ABB RAPID module: 00417E3D

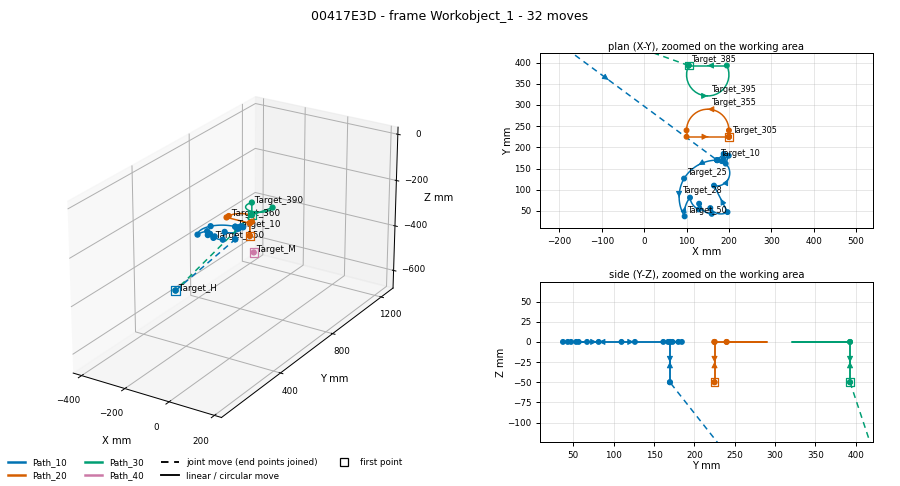
[picture p0: tool path of 00417E3D in frame Workobject_1, 32 of 32 moves have a stored position in this frame; points joined in program order, loops and branches not executed]
MODULE Module1
        CONST robtarget Target_H:=[[-349.999997471,555.651291784,-538.588637673],[0.701057388,-0.092295986,-0.092295969,-0.701057375],[0,0,0,0],[9E+09,9E+09,9E+09,9E+09,9E+09,9E+09]];
    CONST robtarget Target_10:=[[172.145654378,169.721037846,0],[0.015654757,0,0,0.999877457],[1,-2,1,0],[9E+09,9E+09,9E+09,9E+09,9E+09,9E+09]];
    CONST robtarget Target_20:=[[127.176015411,158.806349071,0],[0.015654757,0,0,0.999877457],[1,-2,1,0],[9E+09,9E+09,9E+09,9E+09,9E+09,9E+09]];
    CONST robtarget Target_30:=[[94.179068929,126.362545613,0],[0.015654757,0,0,0.999877457],[1,-2,1,0],[9E+09,9E+09,9E+09,9E+09,9E+09,9E+09]];
    CONST robtarget Target_40:=[[82.505775243,81.583833322,0],[0.015654757,0,0,0.999877457],[1,-2,1,0],[9E+09,9E+09,9E+09,9E+09,9E+09,9E+09]];
    CONST robtarget Target_50:=[[95.464213358,37.159991282,0],[0.015654757,0,0,0.999877457],[1,-2,1,0],[9E+09,9E+09,9E+09,9E+09,9E+09,9E+09]];
    CONST robtarget Target_60:=[[108.140548997,81.368919049,0],[0.015654757,0,0,0.999877457],[1,-2,1,0],[9E+09,9E+09,9E+09,9E+09,9E+09,9E+09]];
    CONST robtarget Target_70:=[[99.986563128,67.9517476,0],[0.015654757,0,0,0.999877457],[1,-2,1,0],[9E+09,9E+09,9E+09,9E+09,9E+09,9E+09]];
    CONST robtarget Target_80:=[[115.844,63.278,0],[0.015654757,0,0,0.999877457],[1,-2,1,0],[9E+09,9E+09,9E+09,9E+09,9E+09,9E+09]];
    CONST robtarget Target_90:=[[110.943419364,69.425655071,0],[0.015654757,0,0,0.999877457],[1,-2,1,0],[9E+09,9E+09,9E+09,9E+09,9E+09,9E+09]];
    CONST robtarget Target_100:=[[118.270530204,59.586392727,0],[0.015654757,0,0,0.999877457],[1,-2,1,0],[9E+09,9E+09,9E+09,9E+09,9E+09,9E+09]];
    CONST robtarget Target_110:=[[128.909818396,53.478759508,0],[0.015654757,0,0,0.999877457],[1,-2,1,0],[9E+09,9E+09,9E+09,9E+09,9E+09,9E+09]];
    CONST robtarget Target_120:=[[129.685602376,67.032677318,0],[0.015654757,0,0,0.999877457],[1,-2,1,0],[9E+09,9E+09,9E+09,9E+09,9E+09,9E+09]];
    CONST robtarget Target_130:=[[135.242270658,54.463630271,0],[0.015654757,0,0,0.999877457],[1,-2,1,0],[9E+09,9E+09,9E+09,9E+09,9E+09,9E+09]];
    CONST robtarget Target_140:=[[145.944316156,45.842509218,0],[0.015654757,0,0,0.999877457],[1,-2,1,0],[9E+09,9E+09,9E+09,9E+09,9E+09,9E+09]];
    CONST robtarget Target_150:=[[159.408253951,43.089350102,0],[0.015654757,0,0,0.999877457],[1,-2,1,0],[9E+09,9E+09,9E+09,9E+09,9E+09,9E+09]];
    CONST robtarget Target_160:=[[156.13873613,56.659281011,0],[0.015654757,0,0,0.999877457],[1,-2,1,0],[9E+09,9E+09,9E+09,9E+09,9E+09,9E+09]];
    CONST robtarget Target_170:=[[167.339659667,46.46756084,0],[0.015654757,0,0,0.999877457],[1,-2,1,0],[9E+09,9E+09,9E+09,9E+09,9E+09,9E+09]];
    CONST robtarget Target_180:=[[156.961,49.601,0],[0.015654757,0,0,0.999877457],[1,-2,1,0],[9E+09,9E+09,9E+09,9E+09,9E+09,9E+09]];
    CONST robtarget Target_190:=[[196.643218036,47.197896671,0],[0.015654757,0,0,0.999877457],[1,-1,1,0],[9E+09,9E+09,9E+09,9E+09,9E+09,9E+09]];
    CONST robtarget Target_200:=[[180.134939682,64.681155269,0],[0.015654757,0,0,0.999877457],[1,-2,1,0],[9E+09,9E+09,9E+09,9E+09,9E+09,9E+09]];
    CONST robtarget Target_210:=[[169.208263421,86.100663464,0],[0.015654757,0,0,0.999877457],[1,-2,1,0],[9E+09,9E+09,9E+09,9E+09,9E+09,9E+09]];
    CONST robtarget Target_220:=[[164.744756678,109.728289095,0],[0.015654757,0,0,0.999877457],[1,-2,1,0],[9E+09,9E+09,9E+09,9E+09,9E+09,9E+09]];
    CONST robtarget Target_230:=[[189.86479429,115.046784411,0],[0.015654757,0,0,0.999877457],[1,-2,1,0],[9E+09,9E+09,9E+09,9E+09,9E+09,9E+09]];
    CONST robtarget Target_240:=[[201.945805105,137.70405388,0],[0.015654757,0,0,0.999877457],[1,-2,1,0],[9E+09,9E+09,9E+09,9E+09,9E+09,9E+09]];
    CONST robtarget Target_250:=[[192.36364797,161.525996428,0],[0.015654757,0,0,0.999877457],[1,-2,1,0],[9E+09,9E+09,9E+09,9E+09,9E+09,9E+09]];
    CONST robtarget Target_260:=[[199.538662434,180.200691671,0],[0.015654757,0,0,0.999877457],[1,-2,1,0],[9E+09,9E+09,9E+09,9E+09,9E+09,9E+09]];
    CONST robtarget Target_270:=[[187.501772235,172.981329375,0],[0.015654757,0,0,0.999877457],[1,-2,1,0],[9E+09,9E+09,9E+09,9E+09,9E+09,9E+09]];
    CONST robtarget Target_280:=[[183.067776679,167.478919652,0],[0.015654757,0,0,0.999877457],[1,-2,1,0],[9E+09,9E+09,9E+09,9E+09,9E+09,9E+09]];
    CONST robtarget Target_290:=[[187.548582623,184.533188144,0],[0.015654757,0,0,0.999877457],[1,-2,1,0],[9E+09,9E+09,9E+09,9E+09,9E+09,9E+09]];
    CONST robtarget Target_300:=[[172.145654378,169.721037846,0],[0.015654757,0,0,0.999877457],[1,-2,1,0],[9E+09,9E+09,9E+09,9E+09,9E+09,9E+09]];
    CONST robtarget Target_305:=[[200,225,-50],[0.015654757,0,0,0.999877457],[1,-2,1,0],[9E+09,9E+09,9E+09,9E+09,9E+09,9E+09]];
    CONST robtarget Target_310:=[[200,225,0],[0.015654757,0,0,0.999877457],[1,-2,1,0],[9E+09,9E+09,9E+09,9E+09,9E+09,9E+09]];
    CONST robtarget Target_320:=[[200,240,0],[0.015654757,0,0,0.999877457],[1,-2,1,0],[9E+09,9E+09,9E+09,9E+09,9E+09,9E+09]];
    CONST robtarget Target_330:=[[185.355339059,275.355339059,0],[0.015654757,0,0,0.999877457],[1,-2,1,0],[9E+09,9E+09,9E+09,9E+09,9E+09,9E+09]];
    CONST robtarget Target_340:=[[150,290,0],[0.015654757,0,0,0.999877457],[1,-2,1,0],[9E+09,9E+09,9E+09,9E+09,9E+09,9E+09]];
    CONST robtarget Target_350:=[[114.644660941,275.355339059,0],[0.015654757,0,0,0.999877457],[1,-2,1,0],[9E+09,9E+09,9E+09,9E+09,9E+09,9E+09]];
    CONST robtarget Target_360:=[[100,240,0],[0.015654757,0,0,0.999877457],[1,-2,1,0],[9E+09,9E+09,9E+09,9E+09,9E+09,9E+09]];
    CONST robtarget Target_370:=[[100,225,0],[0.015654757,0,0,0.999877457],[1,-2,1,0],[9E+09,9E+09,9E+09,9E+09,9E+09,9E+09]];
    CONST robtarget Target_380:=[[200,225,0],[0.015654757,0,0,0.999877457],[1,-2,1,0],[9E+09,9E+09,9E+09,9E+09,9E+09,9E+09]];
    CONST robtarget Target_385:=[[105,392.991805459,-50],[0.015654757,0,0,0.999877457],[1,-2,1,0],[9E+09,9E+09,9E+09,9E+09,9E+09,9E+09]];
    CONST robtarget Target_390:=[[105,392.991805459,0],[0.015654757,0,0,0.999877457],[1,-2,1,0],[9E+09,9E+09,9E+09,9E+09,9E+09,9E+09]];
    CONST robtarget Target_400:=[[103.164813866,353.691159257,0],[0.015654757,0,0,0.999877457],[1,-2,1,0],[9E+09,9E+09,9E+09,9E+09,9E+09,9E+09]];
    CONST robtarget Target_410:=[[130.328264565,325.22968273,0],[0.015654757,0,0,0.999877457],[1,-2,1,0],[9E+09,9E+09,9E+09,9E+09,9E+09,9E+09]];
    CONST robtarget Target_420:=[[169.671735435,325.22968273,0],[0.015654757,0,0,0.999877457],[1,-2,1,0],[9E+09,9E+09,9E+09,9E+09,9E+09,9E+09]];
    CONST robtarget Target_430:=[[196.835186134,353.691159257,0],[0.015654757,0,0,0.999877457],[1,-2,1,0],[9E+09,9E+09,9E+09,9E+09,9E+09,9E+09]];
    CONST robtarget Target_440:=[[195,392.991805459,0],[0.015654757,0,0,0.999877457],[1,-2,1,0],[9E+09,9E+09,9E+09,9E+09,9E+09,9E+09]];
    CONST robtarget Target_M:=[[-410.514648889,1245.713795009,-649.374024814],[0.613768807,0.08026289,-0.406843498,-0.671806585],[0,-1,0,0],[9E+09,9E+09,9E+09,9E+09,9E+09,9E+09]];
    CONST robtarget Target_355:=[[150,290,0],[0.015654757,0,0,0.999877457],[1,-2,1,0],[9E+09,9E+09,9E+09,9E+09,9E+09,9E+09]];
    CONST robtarget Target_15:=[[127.992,158.531,0],[0.015654757,0,0,0.999877457],[1,-2,1,0],[9E+09,9E+09,9E+09,9E+09,9E+09,9E+09]];
    CONST robtarget Target_28:=[[82.508,84.221,0],[0.015654757,0,0,0.999877457],[1,-2,1,0],[9E+09,9E+09,9E+09,9E+09,9E+09,9E+09]];
    CONST robtarget Target_25:=[[94.179,126.363,0],[0.015654757,0,0,0.999877457],[1,-2,1,0],[9E+09,9E+09,9E+09,9E+09,9E+09,9E+09]];
    CONST robtarget Target_395:=[[150,321.197,0],[0.015654757,0,0,0.999877457],[1,-2,1,0],[9E+09,9E+09,9E+09,9E+09,9E+09,9E+09]];
    CONST robtarget Target_55:=[[97.319,60.55,0],[0.015654757,0,0,0.999877457],[1,-2,1,0],[9E+09,9E+09,9E+09,9E+09,9E+09,9E+09]];
    CONST robtarget Target_125:=[[138.21,52.221,0],[0.015654757,0,0,0.999877457],[1,-2,1,0],[9E+09,9E+09,9E+09,9E+09,9E+09,9E+09]];
    CONST robtarget Target_185:=[[167.277,46.352,0],[0.015654757,0,0,0.999877457],[1,-2,1,0],[9E+09,9E+09,9E+09,9E+09,9E+09,9E+09]];
    CONST robtarget Target_115:=[[128.566,60.282,0],[0.015654757,0,0,0.999877457],[0,0,0,0],[9E+09,9E+09,9E+09,9E+09,9E+09,9E+09]];
!***********************************************************
    !
    ! M?dulo:  Module1
    !
    ! Descripción:
    !   <Introduzca la descripción aquí>
    !
    ! Autor: ASUS
    !
    ! Versión: 1.0
    !
    !***********************************************************


    !***********************************************************
    !
    ! Procedimiento Main
    !
    !   Este es el punto de entrada de su programa
    !
    !***********************************************************
    PROC main()
        !Add your code here
        WHILE TRUE DO
            IF DI_01=1 THEN
                set DO_01;
                first;
                Reset DO_01;
            ELSEIF DI_02=1 THEN
                set DO_02;
                Path_40;
                Reset DO_02;
            ENDIF
        ENDWHILE
    ENDPROC
    PROC Path_10()
        MoveJ Target_H,v100,z5,THerramienta\WObj:=Workobject_1;
        MoveJ [[172.145654378,169.721037846,-50],[0.015654757,0,0,0.999877457],[1,-2,1,0],[9E+09,9E+09,9E+09,9E+09,9E+09,9E+09]],v400,z5,THerramienta\WObj:=Workobject_1;
        MoveL Target_10,v200,z0,THerramienta\WObj:=Workobject_1;
        MoveC Target_15,Target_25,v200,z5,THerramienta\WObj:=Workobject_1;
        MoveC Target_28,Target_50,v200,z0,THerramienta\WObj:=Workobject_1;
        MoveC Target_55,Target_60,v200,z0,THerramienta\WObj:=Workobject_1;
        MoveC Target_80,Target_110,v200,z0,THerramienta\WObj:=Workobject_1;
        MoveC Target_115,Target_120,v200,z0,THerramienta\WObj:=Workobject_1;
        MoveC Target_125,Target_150,v200,z0,THerramienta\WObj:=Workobject_1;
        MoveC Target_180,Target_160,v200,z5,THerramienta\WObj:=Workobject_1;
        MoveC Target_185,Target_190,v200,z5,THerramienta\WObj:=Workobject_1;
        MoveL Target_220,v200,z5,THerramienta\WObj:=Workobject_1;
        MoveC Target_240,Target_250,v200,z5,THerramienta\WObj:=Workobject_1;
        MoveL Target_260,v200,z5,THerramienta\WObj:=Workobject_1;
        MoveL Target_270,v200,z5,THerramienta\WObj:=Workobject_1;
        MoveL Target_280,v200,z5,THerramienta\WObj:=Workobject_1;
        MoveL Target_290,v200,z5,THerramienta\WObj:=Workobject_1;
        MoveL Target_300,v200,z0,THerramienta\WObj:=Workobject_1;
        MoveL [[172.145654378,169.721037846,-50],[0.015654757,0,0,0.999877457],[1,-2,1,0],[9E+09,9E+09,9E+09,9E+09,9E+09,9E+09]],v200,z100,THerramienta\WObj:=Workobject_1;
    ENDPROC
    PROC Path_20()
        MoveJ Target_305,v400,z5,THerramienta\WObj:=Workobject_1;
        MoveL Target_310,v200,z0,THerramienta\WObj:=Workobject_1;
        MoveL Target_320,v200,z5,THerramienta\WObj:=Workobject_1;
        MoveC Target_355,Target_360,v200,z5,THerramienta\WObj:=Workobject_1;
        MoveL Target_370,v200,z5,THerramienta\WObj:=Workobject_1;
        MoveL Target_380,v200,z0,THerramienta\WObj:=Workobject_1;
        MoveL Target_305,v200,z5,THerramienta\WObj:=Workobject_1;
    ENDPROC
    PROC first()
        Path_10;
        Path_20;
        Path_30;
    ENDPROC
    PROC Path_30()
        MoveL Target_385,v200,z5,THerramienta\WObj:=Workobject_1;
        MoveL Target_390,v200,z5,THerramienta\WObj:=Workobject_1;
        MoveC Target_395,Target_440,v200,z5,THerramienta\WObj:=Workobject_1;
        MoveL Target_385,v200,z5,THerramienta\WObj:=Workobject_1;
        MoveJ Target_H,v600,z5,THerramienta\WObj:=Workobject_1;
    ENDPROC
    PROC Path_40()
        MoveJ Target_M,v100,z5,THerramienta\WObj:=Workobject_1;
    ENDPROC
ENDMODULE
